// Mitsubishi GX Works2 project: 2023-04-20 #1   PLC: Q03UDV

// global labels: Global1
VAR_GLOBAL
  PB1 AT X0 : BOOL;
  PB2 AT X1 : BOOL;
  정지 AT X2 : BOOL;
  공급후진 AT X3 : BOOL;
  공급전진 AT X4 : BOOL;
  가공후진 AT X5 : BOOL;
  가공전진 AT X6 : BOOL;
  송출후진 AT X7 : BOOL;
  송출전진 AT X8 : BOOL;
  배출후진 AT X9 : BOOL;
  배출전진 AT X0A : BOOL;
  매거진 AT X0B : BOOL;
  가공센서 AT X0C : BOOL;
  송출센서 AT X0D : BOOL;
  비금속센서 AT X0E : BOOL;
  금속센서 AT X0F : BOOL;
  적색 AT Y20 : BOOL;
  황색 AT Y21 : BOOL;
  녹색 AT Y22 : BOOL;
  공급1 AT Y23 : BOOL;
  공급2 AT Y24 : BOOL;
  가공 AT Y25 : BOOL;
  드릴 AT Y26 : BOOL;
  송출 AT Y27 : BOOL;
  배출 AT Y28 : BOOL;
  컨베이어 AT Y29 : BOOL;
  PB3 AT X10 : BOOL;
END_VAR

PROGRAM 기본동작
VAR
  STATE : INT;
END_VAR
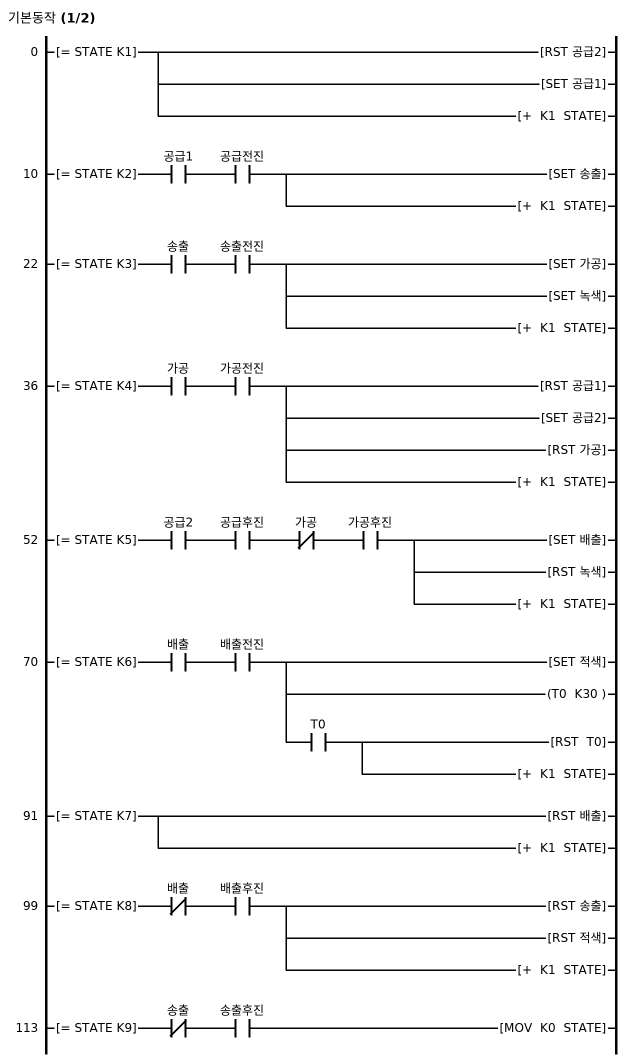
0     LD=     STATE K1
      RST     공급2
      SET     공급1
      +       K1 STATE
10    LD=     STATE K2
      AND     공급1
      AND     공급전진
      SET     송출
      +       K1 STATE
22    LD=     STATE K3
      AND     송출
      AND     송출전진
      SET     가공
      SET     녹색
      +       K1 STATE
36    LD=     STATE K4
      AND     가공
      AND     가공전진
      RST     공급1
      SET     공급2
      RST     가공
      +       K1 STATE
52    LD=     STATE K5
      AND     공급2
      AND     공급후진
      ANI     가공
      AND     가공후진
      SET     배출
      RST     녹색
      +       K1 STATE
70    LD=     STATE K6
      AND     배출
      AND     배출전진
      SET     적색
      OUT     T0 K30
      AND     T0
      RST     T0
      +       K1 STATE
91    LD=     STATE K7
      RST     배출
      +       K1 STATE
99    LD=     STATE K8
      ANI     배출
      AND     배출후진
      RST     송출
      RST     적색
      +       K1 STATE
113   LD=     STATE K9
      ANI     송출
      AND     송출후진
      MOV     K0 STATE
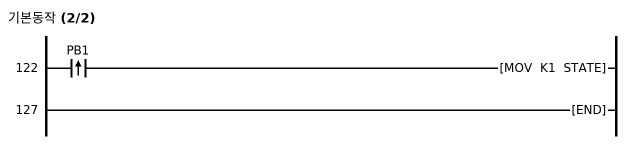
122   LDP     PB1
      MOV     K1 STATE
127   END
END_PROGRAM

PROGRAM 응용동작1
VAR
  STATE : INT;
END_VAR
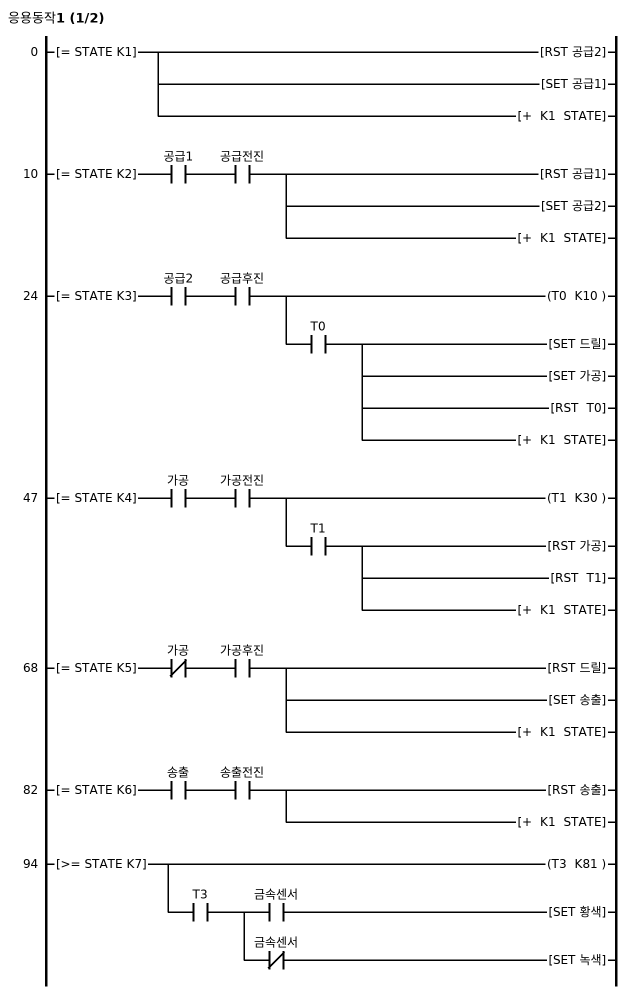
0     LD=     STATE K1
      RST     공급2
      SET     공급1
      +       K1 STATE
10    LD=     STATE K2
      AND     공급1
      AND     공급전진
      RST     공급1
      SET     공급2
      +       K1 STATE
24    LD=     STATE K3
      AND     공급2
      AND     공급후진
      OUT     T0 K10
      AND     T0
      SET     드릴
      SET     가공
      RST     T0
      +       K1 STATE
47    LD=     STATE K4
      AND     가공
      AND     가공전진
      OUT     T1 K30
      AND     T1
      RST     가공
      RST     T1
      +       K1 STATE
68    LD=     STATE K5
      ANI     가공
      AND     가공후진
      RST     드릴
      SET     송출
      +       K1 STATE
82    LD=     STATE K6
      AND     송출
      AND     송출전진
      RST     송출
      +       K1 STATE
94    LD>=    STATE K7
      OUT     T3 K81
      AND     T3
      MPS
      AND     금속센서
      SET     황색
      MPP
      ANI     금속센서
      SET     녹색
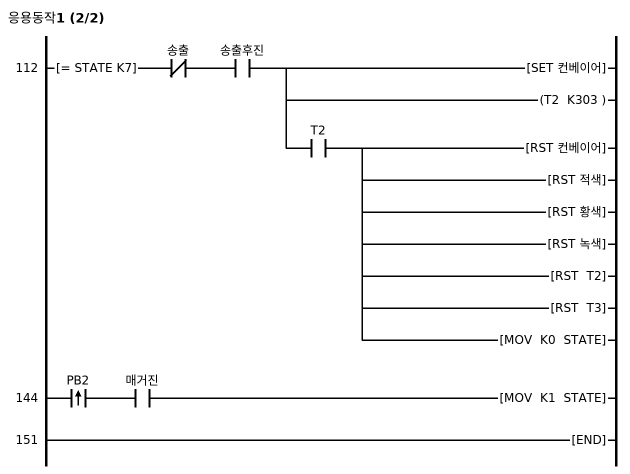
112   LD=     STATE K7
      ANI     송출
      AND     송출후진
      SET     컨베이어
      OUT     T2 K303
      AND     T2
      RST     컨베이어
      RST     적색
      RST     황색
      RST     녹색
      RST     T2
      RST     T3
      MOV     K0 STATE
144   LDP     PB2
      AND     매거진
      MOV     K1 STATE
151   END
END_PROGRAM

PROGRAM 응용동작2
VAR
  STATE : INT;
  STATE2 : INT;
  COUNT : INT;
  COUNT2 : INT;
END_VAR
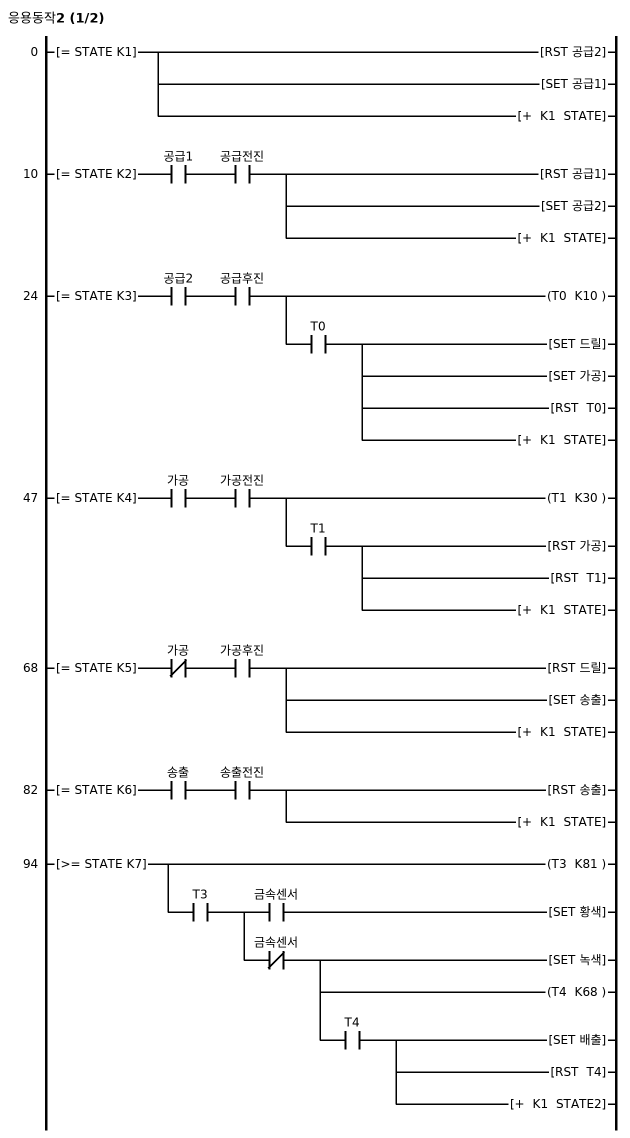
0     LD=     STATE K1
      RST     공급2
      SET     공급1
      +       K1 STATE
10    LD=     STATE K2
      AND     공급1
      AND     공급전진
      RST     공급1
      SET     공급2
      +       K1 STATE
24    LD=     STATE K3
      AND     공급2
      AND     공급후진
      OUT     T0 K10
      AND     T0
      SET     드릴
      SET     가공
      RST     T0
      +       K1 STATE
47    LD=     STATE K4
      AND     가공
      AND     가공전진
      OUT     T1 K30
      AND     T1
      RST     가공
      RST     T1
      +       K1 STATE
68    LD=     STATE K5
      ANI     가공
      AND     가공후진
      RST     드릴
      SET     송출
      +       K1 STATE
82    LD=     STATE K6
      AND     송출
      AND     송출전진
      RST     송출
      +       K1 STATE
94    LD>=    STATE K7
      OUT     T3 K81
      AND     T3
      MPS
      AND     금속센서
      SET     황색
      MPP
      ANI     금속센서
      SET     녹색
      OUT     T4 K68
      AND     T4
      SET     배출
      RST     T4
      +       K1 STATE2
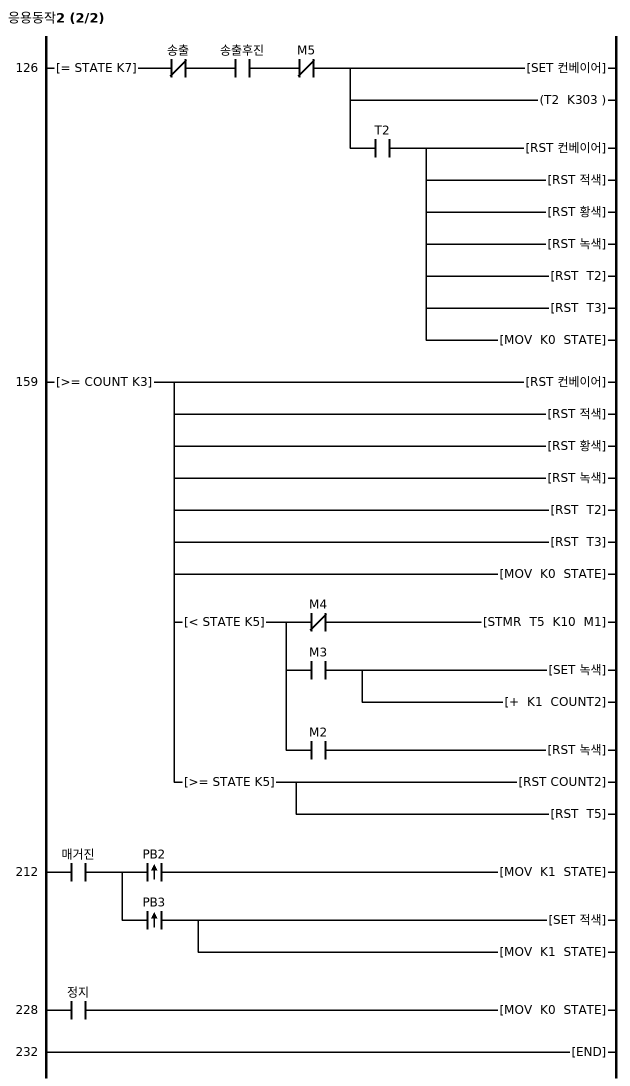
126   LD=     STATE K7
      ANI     송출
      AND     송출후진
      ANI     M5
      SET     컨베이어
      OUT     T2 K303
      AND     T2
      RST     컨베이어
      RST     적색
      RST     황색
      RST     녹색
      RST     T2
      RST     T3
      MOV     K0 STATE
159   LD>=    COUNT K3
      RST     컨베이어
      RST     적색
      RST     황색
      RST     녹색
      RST     T2
      RST     T3
      MOV     K0 STATE
      MPS
      AND<    STATE K5
      MPS
      ANI     M4
      STMR    T5 K10 M1
      MRD
      AND     M3
      SET     녹색
      +       K1 COUNT2
      MPP
      AND     M2
      RST     녹색
      MPP
      AND>=   STATE K5
      RST     COUNT2
      RST     T5
212   LD      매거진
      MPS
      ANDP    PB2
      MOV     K1 STATE
      MPP
      ANDP    PB3
      SET     적색
      MOV     K1 STATE
228   LD      정지
      MOV     K0 STATE
232   END
END_PROGRAM
